INTERFACE I_JsonTypeConverters

METHOD PUBLIC GetByDataType : I_JsonTypeConverter
VAR_INPUT
	DataType : T_MAXSTRING;
END_VAR
END_METHOD

METHOD PUBLIC HasDataType : BOOL
VAR_INPUT
	DataType : T_MAXSTRING;
END_VAR
END_METHOD

METHOD PUBLIC InsertByDataType
VAR_INPUT
	DataType : T_MAXSTRING;
	TypeConverter : I_JsonTypeConverter;
END_VAR
END_METHOD

END_INTERFACE

(* stored: Version 1.1.0.1, ProductVersion 3.1.4024.12
   Itf I_JsonTypeConverters: Id {f77e546c-bf53-07d4-014d-a227dc9dfa40}
   Method GetByDataType: Id {ee358f18-488f-0191-2e49-1323b9f70ae1}
   Method HasDataType: Id {f0da7e27-5e99-0091-2da9-2bec43aa526d}
   Method InsertByDataType: Id {361fcd9d-d264-0365-2cf9-c9886efb0859} *)
